FUNCTION_BLOCK I_TD_TD (* ISOBUS Time/Date Wrapper with TD Struct Output *)
  (* Standard: ISO 11783-7; Classification: PGN 65254; Description: Copyright (c) 2024-2026 HR Agrartechnik GmbH This program and the accompanying materials are made available under the terms of the Eclipse Public License 2.0 which is available at https://www.eclipse.org/legal/epl-2.0/ SPDX-License-Identifier: EPL-2.0 Wrapper around I_TD providing time/date as TD struct. https://docs.ms-muc-docs.de/projects/isobus-other-docs/de/latest/PGN/PGN_65254.html *)
  (* Version 1.0, 2026-04-24, Franz Höpfinger, HR Agrartechnik GmbH, Wrapper combining time/date components into TD struct *)
  PACKAGE isobus::tecu;
  IMPORT eclipse4diac::core::TypeHash;
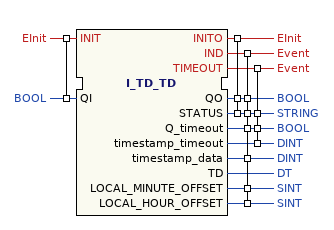
  EVENT_INPUT
    INIT : EInit WITH QI; (* Service Initialization *)
  END_EVENT
  EVENT_OUTPUT
    INITO : EInit WITH QO, STATUS; (* Initialization Confirm *)
    IND WITH QO, timestamp_data, STATUS, Q_timeout, LOCAL_MINUTE_OFFSET, LOCAL_HOUR_OFFSET; (* Indication from Resource *)
    TIMEOUT WITH timestamp_timeout, STATUS, Q_timeout;
  END_EVENT
  VAR_INPUT
    QI : BOOL; (* Event Input Qualifier *)
  END_VAR
  VAR_OUTPUT
    QO : BOOL; (* Event Output Qualifier *)
    STATUS : STRING;
    Q_timeout : BOOL;
    timestamp_timeout : DINT;
    timestamp_data : DINT;
    TD : DT; (* Time/Date as defined in IEC 61131-3 *)
    LOCAL_MINUTE_OFFSET : SINT; (* Local minute offset (see Attributes for Details) *) {SET_ATTRIBUTE(SPN, 1601)} {SET_ATTRIBUTE(SP_Name, 'Local minute offset')} {SET_ATTRIBUTE(SP_Position_In_PG, '7')} {SET_ATTRIBUTE(SP_Length, 8)} (* 8 bits *) {SET_ATTRIBUTE(Scaling, '1 min/bit')} {SET_ATTRIBUTE(Offset, -125)} {SET_ATTRIBUTE(Link, 'https://docs.ms-muc-docs.de/projects/isobus-other-docs/de/latest/PGN/PGN_65254.html#spn-1601-local-minute-offset')}
    LOCAL_HOUR_OFFSET : SINT; (* Local hour offset (see Attributes for Details) *) {SET_ATTRIBUTE(SPN, 1602)} {SET_ATTRIBUTE(SP_Name, 'Local hour offset')} {SET_ATTRIBUTE(SP_Position_In_PG, '8')} {SET_ATTRIBUTE(SP_Length, 8)} (* 8 bits *) {SET_ATTRIBUTE(Scaling, '1 h/bit')} {SET_ATTRIBUTE(Offset, -125)} {SET_ATTRIBUTE(Link, 'https://docs.ms-muc-docs.de/projects/isobus-other-docs/de/latest/PGN/PGN_65254.html#spn-1602-local-hour-offset')}
  END_VAR
  FBS
    I_CORE : isobus::tecu::I_TD;
    F_CONCAT_DT : iec61131::charString::F_CONCAT_DT;
  END_FBS
  EVENT_CONNECTIONS
    INIT TO I_CORE.INIT;
    I_CORE.INITO TO INITO;
    I_CORE.TIMEOUT TO TIMEOUT;
    I_CORE.IND TO F_CONCAT_DT.REQ;
    F_CONCAT_DT.CNF TO IND;
  END_CONNECTIONS
  DATA_CONNECTIONS
    QI TO I_CORE.QI;
    I_CORE.QO TO QO;
    I_CORE.STATUS TO STATUS;
    I_CORE.Q_timeout TO Q_timeout;
    I_CORE.LOCAL_MINUTE_OFFSET TO LOCAL_MINUTE_OFFSET;
    I_CORE.LOCAL_HOUR_OFFSET TO LOCAL_HOUR_OFFSET;
    I_CORE.timestamp_timeout TO timestamp_timeout;
    I_CORE.timestamp_data TO timestamp_data;
    I_CORE.YEAR TO F_CONCAT_DT.YEAR;
    I_CORE.MONTH TO F_CONCAT_DT.MONTH;
    I_CORE.DAY TO F_CONCAT_DT.DAY;
    I_CORE.HOURS TO F_CONCAT_DT.HOUR;
    I_CORE.MINUTES TO F_CONCAT_DT.MINUTE;
    I_CORE.SECONDS TO F_CONCAT_DT.SECOND;
    F_CONCAT_DT.OUT TO TD;
  END_CONNECTIONS
END_FUNCTION_BLOCK
